ABB RobotStudio station: Solution_1.rspag

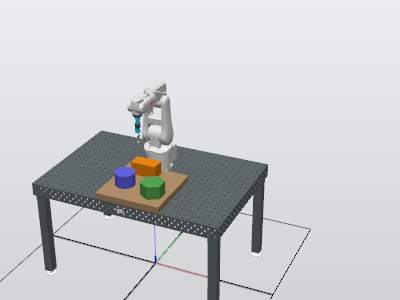
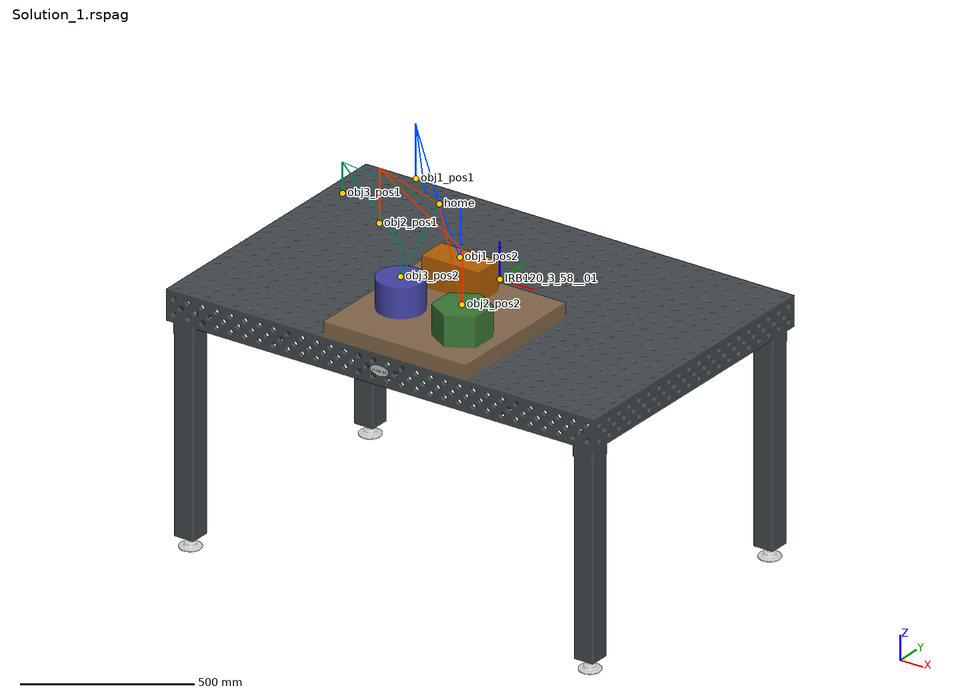
[picture v1: parts stored in the station drawn from their meshes, with robot base, taught points and paths (robot models come from the ABB library and are not in the file)]
--- station ---
Station Solution_1_Tutorial (saved by RobotStudio 22.3.10190.2)
Controller Controller1, task T_ROB1: task frame (RAPID world) sits at (0, 100, 830) mm, rotated rx 0 ry 0 rz -90 deg in the station
Controller Controller1
  mechanical unit ROB_1: IRB120_3_58__01, 6 joints, base frame (0, 0, 0) mm
Layout (positions relative to the parent item):
  - table [part] at (-200, -500, 830) mm, size 500 x 500 x 50 mm
  - object_1 [part] at (-200, -500, 830) mm, size 200 x 100 x 150 mm
  - object_2 [part] at (-200, -500, 830) mm, size 149.5 x 149.7 x 150 mm
  - object_3 [part] at (-200, -500, 830) mm, size 155.5 x 179.5 x 150 mm
  - siegmund_1500_1000 [part], size 1500 x 1010.3 x 830 mm
  - object_11 [part] at (-200, -500, 830) mm, size 200 x 100 x 150 mm
  - object_22 [part] at (-200, -500, 830) mm, size 149.5 x 149.7 x 150 mm
  - object_33 [part] at (-200, -500, 830) mm, size 155.5 x 179.5 x 150 mm
  - IRB120_3_58__01 [mechanism, from Robots\IRB120_3_58_G_01.rslib] at (0, 100, 830) mm, rotated rx 0 ry 0 rz -90 deg; joint values [0, 0, 0, 0, 1.5708, 0] (rad or m)
  - smc_gripper [mechanism, from Libraries\smc_gripper.rslib] at (0, -202, 1388) mm, rotated rx 180 ry 0 rz 90 deg
  - positioner_obj_1 [smart component, from Components\Positioner.rslib]
      properties: Object=object_1; Position=[-0.6 -0.15 0.83]; Orientation=[0 0 0]; Reference=Global; ReferenceObject=(none)
  - Detacher [smart component, from Components\Detacher.rslib]
      properties: Child=object_1; KeepPosition=true
  - Attacher [smart component, from Components\Attacher.rslib]
      properties: Parent=smc_gripper; Flange=0; Child=object_1; Mount=false; Offset=[0 0 0]; Orientation=[0 0 0]
  - Positioner_2 [smart component, from Components\Positioner.rslib] at (-650, -150, 830) mm
      properties: Object=object_3; Position=[-0.7 -0.2 0.83]; Orientation=[0 0 0]; Reference=Global; ReferenceObject=(none)
  - Attacher_2 [smart component, from Components\Attacher.rslib]
      properties: Parent=smc_gripper; Flange=0; Child=object_3; Mount=false; Offset=[0 0 0]; Orientation=[0 0 0]
  - Detacher_2 [smart component, from Components\Detacher.rslib]
      properties: Child=object_3; KeepPosition=true
  - Positioner_3 [smart component, from Components\Positioner.rslib]
      properties: Object=object_2; Position=[-0.65 -0.15 0.83]; Orientation=[0 0 0]; Reference=Global; ReferenceObject=(none)
  - Detacher_3 [smart component, from Components\Detacher.rslib]
      properties: Child=object_2; KeepPosition=true
  - Attacher_3 [smart component, from Components\Attacher.rslib]
      properties: Parent=smc_gripper; Flange=0; Child=object_2; Mount=false; Offset=[0 0 0]; Orientation=[0 0 0]
Attachment: smc_gripper is attached to IRB120_3_58__01 / Link6
Collision set CollisionSet_1: object_1, object_2, object_3 against IRB120_3_58__01, object_3, object_2, object_1, near miss 0 m
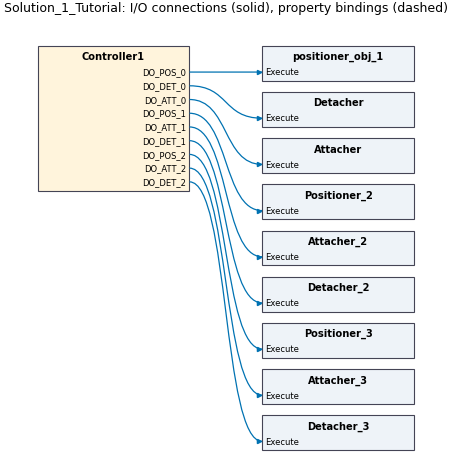
Station logic (signal -> signal, property => property):
  Controller1.DO_POS_0 -> positioner_obj_1.Execute
  Controller1.DO_DET_0 -> Detacher.Execute
  Controller1.DO_ATT_0 -> Attacher.Execute
  Controller1.DO_POS_1 -> Positioner_2.Execute
  Controller1.DO_ATT_1 -> Attacher_2.Execute
  Controller1.DO_DET_1 -> Detacher_2.Execute
  Controller1.DO_POS_2 -> Positioner_3.Execute
  Controller1.DO_ATT_2 -> Attacher_3.Execute
  Controller1.DO_DET_2 -> Detacher_3.Execute

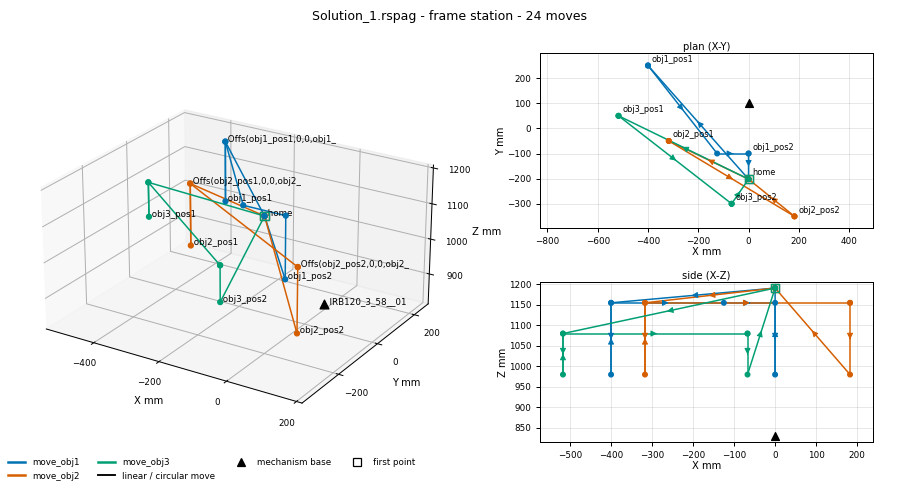
[picture p0: tool path of Solution_1.rspag in frame station, 24 of 24 moves have a stored position in this frame; points joined in program order, loops and branches not executed]
--- Backups/Controller1/RAPID/TASK1/PROGMOD/CalibData.mod ---
MODULE CalibData
    PERS tooldata smc_gripper:=[TRUE,[[0,0.004,197.001],[1,0,0,0]],[1,[0.207,-0.496,71.18],[1,0,0,0],0,0,0]];
ENDMODULE

--- Backups/Controller1/RAPID/TASK1/PROGMOD/Module1.mod ---
MODULE Module1
    CONST robtarget home:=[[302,0.004,360.999],[0,0,1,0],[-1,0,-1,0],[9E+09,9E+09,9E+09,9E+09,9E+09,9E+09]];

    CONST robtarget obj1_pos1:=[[-150,-400,150],[0,0,1,0],[-2,0,-2,0],[9E+09,9E+09,9E+09,9E+09,9E+09,9E+09]];
    CONST robtarget obj1_pos2:=[[200,0,150],[0,0,1,0],[-1,0,-1,0],[9E+09,9E+09,9E+09,9E+09,9E+09,9E+09]];

    CONST robtarget obj2_pos1:=[[150,-317.298,150],[0,0,1,0],[-1,0,-1,0],[9E+09,9E+09,9E+09,9E+09,9E+09,9E+09]];
    CONST robtarget obj2_pos2:=[[450,182.702,150],[0,0,1,0],[0,0,0,0],[9E+09,9E+09,9E+09,9E+09,9E+09,9E+09]];

    CONST robtarget obj3_pos1:=[[50,-517.298,150],[0,0,1,0],[0,0,0,0],[9E+09,9E+09,9E+09,9E+09,9E+09,9E+09]];
    CONST robtarget obj3_pos2:=[[400,-67.298,150],[0,0,1,0],[0,0,0,0],[9E+09,9E+09,9E+09,9E+09,9E+09,9E+09]];

    VAR num obj1_offset_z := 175;
    VAR num obj2_offset_z := 175;
    VAR num obj3_offset_z := 100;
    VAR num obj1_offset_y := -125;

    PROC main()
        init_obj_position;
        move_obj1;
        move_obj2;
        move_obj3;
    ENDPROC

    PROC init_obj_position()
        PulseDO DO_POS_0;
        PulseDO DO_POS_1;
        PulseDO DO_POS_2;
    ENDPROC

    PROC move_obj1()
        MoveL home,v500,fine,smc_gripper\WObj:=wobj0;
        MoveL Offs(obj1_pos1, 0, 0, obj1_offset_z),v500,z100,smc_gripper\WObj:=wobj0;
        MoveL obj1_pos1,v500,fine,smc_gripper\WObj:=wobj0;
        WaitTime 0.5;
        PulseDO DO_ATT_0;
        MoveL Offs(obj1_pos1, 0, 0, obj1_offset_z),v500,z100,smc_gripper\WObj:=wobj0;
        MoveL Offs(obj1_pos2, 0, obj1_offset_y, obj1_offset_z),v500,fine,smc_gripper\WObj:=wobj0;
        MoveL Offs(obj1_pos2, 0, 0, obj1_offset_z),v500,z100,smc_gripper\WObj:=wobj0;
        MoveL obj1_pos2,v500,fine,smc_gripper\WObj:=wobj0;
        WaitTime 0.5;
        PulseDO DO_DET_0;
        MoveL home,v500,fine,smc_gripper\WObj:=wobj0;
    ENDPROC

    PROC move_obj2()
        MoveL home,v500,fine,smc_gripper\WObj:=wobj0;
        MoveL Offs(obj2_pos1, 0, 0, obj2_offset_z),v500,z100,smc_gripper\WObj:=wobj0;
        MoveL obj2_pos1,v500,fine,smc_gripper\WObj:=wobj0;
        WaitTime 0.5;
        PulseDO DO_ATT_1;
        MoveL Offs(obj2_pos1, 0, 0, obj2_offset_z),v500,z100,smc_gripper\WObj:=wobj0;
        MoveL Offs(obj2_pos2, 0, 0, obj2_offset_z),v500,fine,smc_gripper\WObj:=wobj0;
        MoveL Offs(obj2_pos2, 0, 0, obj2_offset_z),v500,z100,smc_gripper\WObj:=wobj0;
        MoveL obj2_pos2,v500,fine,smc_gripper\WObj:=wobj0;
        WaitTime 0.5;
        PulseDO DO_DET_1;
        MoveL home,v500,fine,smc_gripper\WObj:=wobj0;
    ENDPROC

    PROC move_obj3()
        MoveL home,v500,fine,smc_gripper\WObj:=wobj0;
        MoveL Offs(obj3_pos1, 0, 0, obj3_offset_z),v500,z100,smc_gripper\WObj:=wobj0;
        MoveL obj3_pos1,v500,fine,smc_gripper\WObj:=wobj0;
        WaitTime 0.5;
        PulseDO DO_ATT_2;
        MoveL Offs(obj3_pos1, 0, 0, obj3_offset_z),v500,z100,smc_gripper\WObj:=wobj0;
        MoveL Offs(obj3_pos2, 0, 0, obj3_offset_z),v500,fine,smc_gripper\WObj:=wobj0;
        MoveL Offs(obj3_pos2, 0, 0, obj3_offset_z),v500,z100,smc_gripper\WObj:=wobj0;
        MoveL obj3_pos2,v500,fine,smc_gripper\WObj:=wobj0;
        WaitTime 0.5;
        PulseDO DO_DET_2;
        MoveL home,v500,fine,smc_gripper\WObj:=wobj0;
    ENDPROC

ENDMODULE

--- Backups/Controller1/SYSPAR/EIO.cfg ---
EIO:CFG_1.0:6:1::
#
EIO_SIGNAL:

      -Name "DO_POS_0" -SignalType "DO"

      -Name "DO_ATT_0" -SignalType "DO"

      -Name "DO_DET_0" -SignalType "DO"

      -Name "DO_POS_1" -SignalType "DO"

      -Name "DO_DET_1" -SignalType "DO"

      -Name "DO_ATT_1" -SignalType "DO"

      -Name "DO_ATT_2" -SignalType "DO"

      -Name "DO_DET_2" -SignalType "DO"

      -Name "DO_POS_2" -SignalType "DO"
